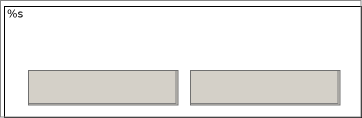
VISUALIZATION VISU_MESSAGE_ALERTE  // 362x118
VAR_IN_OUT
	COM : BLOCK_RS232_ONBOARD_V4;
	var_a_affecter: BOOL:=FALSE;
END_VAR
VAR_INPUT
	valeur_a_affecter: BOOL:=FALSE;
END_VAR
    Rectangle (4,6 358x112), "%s", text list: 'TextList_CryoPump', text index: 89
    Button (28,70 150x35), text list: 'TextList_CryoPump', text index: 92
        OnMouseClick: execute { COM.CO_Envoie_Param_Relay:=true; }
        OnMouseUp: execute { COM.CO_Envoie_Param_Relay:=false; Message_erreur_invisible:=true; }
    Button (190,70 150x35), text list: 'TextList_CryoPump', text index: 93
        OnMouseClick: execute { Message_erreur_invisible:=true; }
    Rectangle (11,30 345x30), text list: 'TextList_CryoPump', text index: 90
END_VISUALIZATION

(* stored: Version 1.1.0.1, ProductVersion 3.1.4026.18
   Visu VISU_MESSAGE_ALERTE: Id {0710b7d5-c941-41b4-98b1-a70196c12df8} *)
